FUNCTION_BLOCK TurnTableManualIReq (* Turn Table Manual Interface Requier *)
  (* Standard: 61499-2 *)
  (* Version 0.2, 2003-12-05, JHC, Rockwell Automation, Renamed from NEWCOMPFB. *)
  (* Version 0.1, 2002-01-08, JHC, Rockwell Automation, Added DLY FB as example. *)
  (* Version 0.0, 2000-05-27, JHC, Rockwell Automation *)
  (* Compiler header: package fb.rt.dasdA1.A2.TurnTable; *)
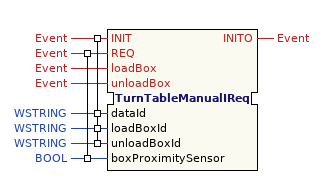
  EVENT_INPUT
    INIT WITH dataId, loadBoxId, unloadBoxId; (* Initialization Request *)
    REQ WITH boxProximitySensor;
    loadBox;
    unloadBox;
  END_EVENT
  EVENT_OUTPUT
    INITO; (* Initialization Confirm *)
  END_EVENT
  VAR_INPUT
    dataId : WSTRING;
    loadBoxId : WSTRING;
    unloadBoxId : WSTRING;
    boxProximitySensor : BOOL;
  END_VAR
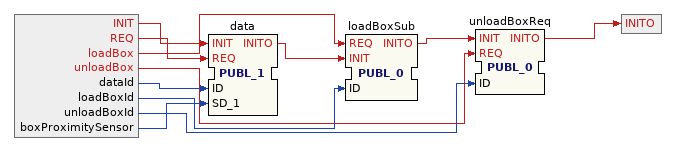
  FBS
    loadBoxSub : PUBL_0;
    data : PUBL_1;
    unloadBoxReq : PUBL_0;
  END_FBS
  EVENT_CONNECTIONS
    loadBox TO loadBoxSub.REQ;
    INIT TO data.INIT;
    REQ TO data.REQ;
    data.INITO TO loadBoxSub.INIT;
    loadBoxSub.INITO TO unloadBoxReq.INIT;
    unloadBoxReq.INITO TO INITO;
    unloadBox TO unloadBoxReq.REQ;
  END_CONNECTIONS
  DATA_CONNECTIONS
    loadBoxId TO loadBoxSub.ID;
    dataId TO data.ID;
    boxProximitySensor TO data.SD_1;
    unloadBoxId TO unloadBoxReq.ID;
  END_CONNECTIONS
END_FUNCTION_BLOCK
